PROGRAM prgMemPointerView
VAR
    pointerToMem:POINTER TO DWORD;  //DWORD
    offset: UDINT; //was UINT
	puls:R_TRIG; //only do stuff sometimes		

	i: INT;
END_VAR
VAR // added by the converter: edge detectors and wires of the graphical bodies
    _rt1, _rt2, _rt3, _rt4 : R_TRIG;
END_VAR

//theme:VyJXkKWsxko

//buttons for adjusting offset, visu is keypad entry
actAdjustOffset();

IF System.PulseOneSecond THEN

	//move offset to keep global
	offset := ioView.memoffset * 4;
	
	//get pointer fata
	actCapturePointer();
	
	//add offset, from 0, add offset to desired memory location, e.g. "0 + 1024 = 1024" to view MD1024 and resulting areas
	pointerToMem := pointerToMem + offset;
	
	CASE ioView.memsize OF
		0://1 bytes per index
		FOR i := 0 TO 15 DO //8bit
			MEMCPY(destAddr:=ADR(ioView.ViewingArray[i]), srcAddr:=pointerToMem + INT_TO_DWORD(i),n:=1);
		END_FOR
		
		1://2 bytes per index
		FOR i := 0 TO 15 DO //16bit
			MEMCPY(destAddr:=ADR(ioView.ViewingArray[i]), srcAddr:=pointerToMem + INT_TO_DWORD(i) * 2,n:=2);
		END_FOR
		
		2://4 bytes per index
		FOR i := 0 TO 15 DO //32bit
			MEMCPY(destAddr:=ADR(ioView.ViewingArray[i]), srcAddr:=pointerToMem + INT_TO_DWORD(i) * 4,n:=4);
		END_FOR
	END_CASE

END_IF

ACTION actAdjustOffset:
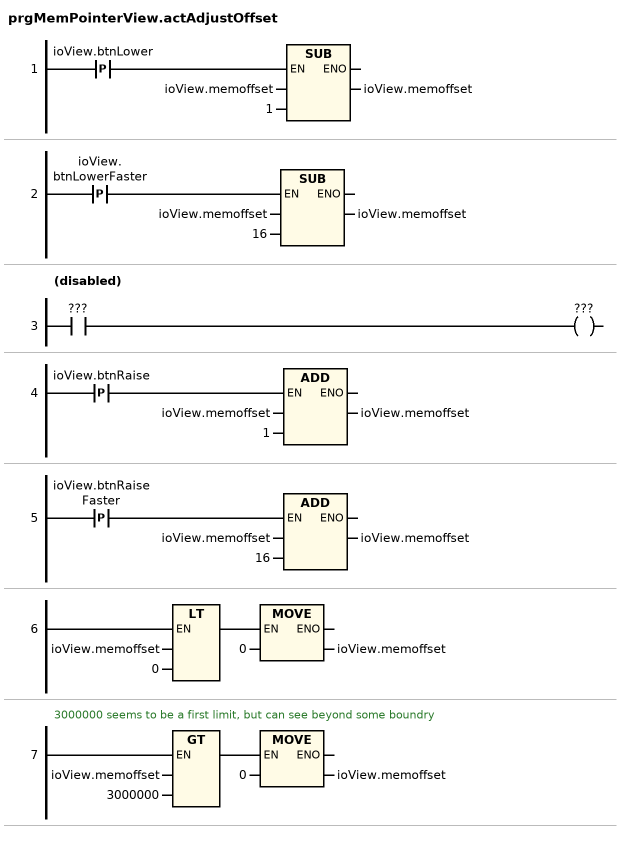
// NETWORK 1
_rt1(CLK := ioView.btnLower);
IF _rt1.Q THEN ioView.memoffset := ioView.memoffset - 1; END_IF

// NETWORK 2
_rt2(CLK := ioView.btnLowerFaster);
IF _rt2.Q THEN ioView.memoffset := ioView.memoffset - 16; END_IF

// NETWORK 3 (disabled)
// ??? := ???;

// NETWORK 4
_rt3(CLK := ioView.btnRaise);
IF _rt3.Q THEN ioView.memoffset := ioView.memoffset + 1; END_IF

// NETWORK 5
_rt4(CLK := ioView.btnRaiseFaster);
IF _rt4.Q THEN ioView.memoffset := ioView.memoffset + 16; END_IF

// NETWORK 6
IF ioView.memoffset < 0 THEN ioView.memoffset := 0; END_IF

// NETWORK 7
// 3000000 seems to be a first limit, but can see beyond some boundry
IF ioView.memoffset > 3000000 THEN ioView.memoffset := 0; END_IF
END_ACTION

ACTION actCapturePointer:
//for M, MEMORY, MD, MW, Mx.y
//theme rbJgtdJLvo8?t=2110	
CASE ioView.memtype OF
	0: //I
	pointerToMem := ADR(%ID0);
	
	1: //Q
	pointerToMem := ADR(%QD0);
	
	2: //M
	pointerToMem := ADR(%MD0);
	
	3: //L
	pointerToMem := ADR(%MD0);
END_CASE
END_ACTION

END_PROGRAM

(* stored: Version 1.1.0.1, ProductVersion 3.1.4024.12
   POU prgMemPointerView: Id {14ad67c0-13ff-42b6-871c-62e51a4859e1}, SpecialFunc None
   Action actAdjustOffset: Id {768519a0-735e-466b-9cc6-26b77674c384}
   Action actCapturePointer: Id {f96964f9-c358-4464-bd11-f7fd4791c184} *)
